// TIA Portal V16 export
// export: Created 2023-03-29T11:04:28.7707464Z, ExportSetting WithDefaults, DisplayName Totally Integrated Automation Portal, DisplayVersion V16 Update 6, DisplayName TIA Portal Version Control Interface, DisplayVersion V16 Update 2, DisplayName TIA Portal Openness, DisplayVersion V16 Update 6, DisplayName STEP 7 Professional, DisplayVersion V16 Update 6, DisplayName STEP 7 Safety, DisplayVersion V16, DisplayName WinCC Advanced, DisplayVersion V16 Update 6
FUNCTION "Konverter_zegarów" : Void   // FC31, LAD
{ S7_Optimized_Access := 'FALSE' }
VERSION : 0.1
// stored: AutoNumber true, IsIECCheckEnabled false, SetENOAutomatically false, UDAEnableTagReadback false
   VAR_INPUT
      HOUR : USInt;   // Zmienna godzina z DTL
      MINUTE : USInt;   // Zmienna minuty z DTL
      SECOND : USInt;   // Zmienne sekundy z DTL
   END_VAR
   VAR_OUTPUT
      Czas_Liczba_conv_Real : Real;   // Liczba przedstawiająca czas 00:00:00 liczbowo 00.0000
      Zegar_H : Int;
      Zegar_M : Int;
      Zegar_S : Int;
   END_VAR
   VAR_TEMP
      zegar_H_pomocnicza : Real;   // pomocnicza do przekształcenia czasu z DLT do Real
      zegar_M_pomocnicza : Real;   // pomocnicza do przekształcenia czasu z DLT do Real
      zegar_S_pomocnicza : Real;   // pomocnicza do przekształcenia czasu z DLT do Real
      zegar_H_Uint : UInt;   // pomocnicza do przekształcenia czasu z DLT do Uint
      zegar_M_Uint : UInt;   // pomocnicza do przekształcenia czasu z DLT do Uint
      zegar_S_Uint : UInt;   // pomocnicza do przekształcenia czasu z DLT do Uint
   END_VAR
BEGIN

REGION Network 1: Wyodrębnienie zegara z danej DTL czasu lokalnego
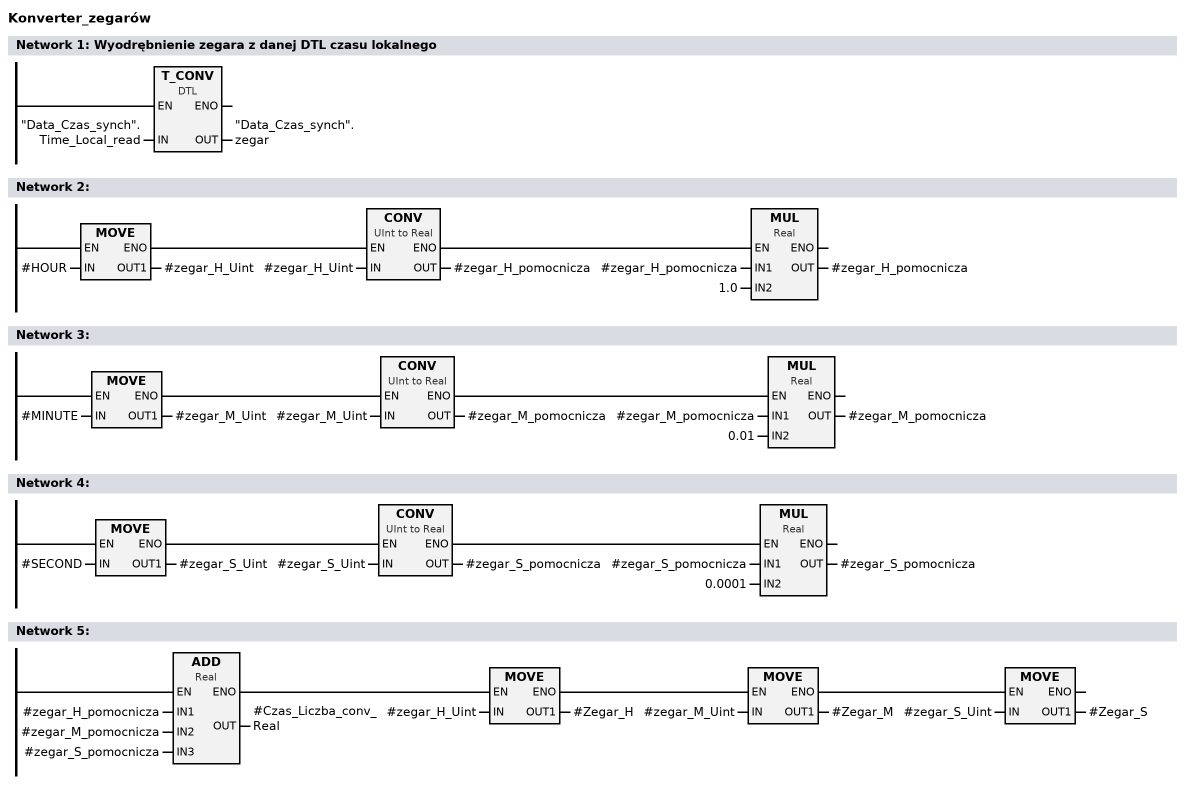
   RUNG wire#powerrail
      { S7_Templates := "[src_type := DTL, dest_type := Time_Of_Day]" } T_CONV(IN := "Data_Czas_synch".Time_Local_read, OUT => "Data_Czas_synch".zegar)
   END_RUNG
   // the same network as SCL:
   T_CONV(IN := "Data_Czas_synch".Time_Local_read, OUT => "Data_Czas_synch".zegar);
END_REGION

REGION Network 2
   RUNG wire#powerrail
      { S7_GenerateENO := "TRUE" } Move(in := #HOUR, out1 => #zegar_H_Uint)
      { S7_Templates := "[SrcType := UInt, DestType := Real]"; S7_GenerateENO := "TRUE" } Convert(in := #zegar_H_Uint, out => #zegar_H_pomocnicza)
      { S7_Templates := "SrcType := Real"; S7_GenerateENO := "TRUE" } Mul(in1 := #zegar_H_pomocnicza, in2 := 1.0, out => #zegar_H_pomocnicza)
   END_RUNG
   // the same network as SCL:
   // ENO of a box is taken as its EN; it also drops when the box reports an error
   #zegar_H_Uint := #HOUR;
   #zegar_H_pomocnicza := UINT_TO_REAL(#zegar_H_Uint);
   #zegar_H_pomocnicza := #zegar_H_pomocnicza * 1.0;
END_REGION

REGION Network 3
   RUNG wire#powerrail
      { S7_GenerateENO := "TRUE" } Move(in := #MINUTE, out1 => #zegar_M_Uint)
      { S7_Templates := "[SrcType := UInt, DestType := Real]"; S7_GenerateENO := "TRUE" } Convert(in := #zegar_M_Uint, out => #zegar_M_pomocnicza)
      { S7_Templates := "SrcType := Real"; S7_GenerateENO := "TRUE" } Mul(in1 := #zegar_M_pomocnicza, in2 := 0.01, out => #zegar_M_pomocnicza)
   END_RUNG
   // the same network as SCL:
   // ENO of a box is taken as its EN; it also drops when the box reports an error
   #zegar_M_Uint := #MINUTE;
   #zegar_M_pomocnicza := UINT_TO_REAL(#zegar_M_Uint);
   #zegar_M_pomocnicza := #zegar_M_pomocnicza * 0.01;
END_REGION

REGION Network 4
   RUNG wire#powerrail
      { S7_GenerateENO := "TRUE" } Move(in := #SECOND, out1 => #zegar_S_Uint)
      { S7_Templates := "[SrcType := UInt, DestType := Real]"; S7_GenerateENO := "TRUE" } Convert(in := #zegar_S_Uint, out => #zegar_S_pomocnicza)
      { S7_Templates := "SrcType := Real"; S7_GenerateENO := "TRUE" } Mul(in1 := #zegar_S_pomocnicza, in2 := 0.0001, out => #zegar_S_pomocnicza)
   END_RUNG
   // the same network as SCL:
   // ENO of a box is taken as its EN; it also drops when the box reports an error
   #zegar_S_Uint := #SECOND;
   #zegar_S_pomocnicza := UINT_TO_REAL(#zegar_S_Uint);
   #zegar_S_pomocnicza := #zegar_S_pomocnicza * 0.0001;
END_REGION

REGION Network 5
   RUNG wire#powerrail
      { S7_Templates := "SrcType := Real"; S7_GenerateENO := "TRUE" } Add(in1 := #zegar_H_pomocnicza, in2 := #zegar_M_pomocnicza, in3 := #zegar_S_pomocnicza, out => #Czas_Liczba_conv_Real)
      Move(in := #zegar_H_Uint, out1 => #Zegar_H)
      Move(in := #zegar_M_Uint, out1 => #Zegar_M)
      Move(in := #zegar_S_Uint, out1 => #Zegar_S)
   END_RUNG
   // the same network as SCL:
   // ENO of a box is taken as its EN; it also drops when the box reports an error
   #Czas_Liczba_conv_Real := #zegar_H_pomocnicza + #zegar_M_pomocnicza + #zegar_S_pomocnicza;
   #Zegar_H := #zegar_H_Uint;
   #Zegar_M := #zegar_M_Uint;
   #Zegar_S := #zegar_S_Uint;
END_REGION
END_FUNCTION
